ADAPTER IMotStatus (* Adapter Interface *)
  (* Standard: 61499-1 *)
  (* Version 0.0, 3/5/2026, Schneider Electric *)
  PACKAGE SE.Nereda;
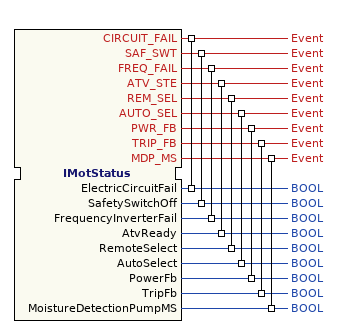
  EVENT_OUTPUT
    CIRCUIT_FAIL WITH ElectricCircuitFail;
    SAF_SWT WITH SafetySwitchOff;
    FREQ_FAIL WITH FrequencyInverterFail;
    ATV_STE WITH AtvReady;
    REM_SEL WITH RemoteSelect;
    AUTO_SEL WITH AutoSelect;
    PWR_FB WITH PowerFb;
    TRIP_FB WITH TripFb;
    MDP_MS WITH MoistureDetectionPumpMS;
  END_EVENT
  VAR_OUTPUT
    ElectricCircuitFail : BOOL;
    SafetySwitchOff : BOOL;
    FrequencyInverterFail : BOOL;
    AtvReady : BOOL;
    RemoteSelect : BOOL;
    AutoSelect : BOOL;
    PowerFb : BOOL;
    TripFb : BOOL;
    MoistureDetectionPumpMS : BOOL;
  END_VAR
  SERVICE SOCKET/PLUG
    SEQUENCE request_confirm
      SOCKET.REQ(REQD) -> PLUG.REQ(REQD);
      PLUG.CNF(CNFD) -> SOCKET.CNF(CNFD);
    END_SEQUENCE
    SEQUENCE indication_response
      PLUG.IND(INDD) -> SOCKET.IND(INDD);
      SOCKET.RSP(RSPD) -> PLUG.RSP(RSPD);
    END_SEQUENCE
  END_SERVICE
END_ADAPTER
